# EPICS autosave request: optics/opticsApp/Db/ml_monoSeq_settings.req
# Multilayer monochromator
$(P)ml_monoD.VAL
$(P)ml_monoOrder.VAL
$(P)ml_monoMode2.VAL
$(P)ml_monoETweak
$(P)ml_monoLambdaTweak
$(P)ml_monoTheta.VAL
